% RSLogix 500 project INVENTORY_MANAGEMENT.RSS, saved by version 8.30.00.16 %
PROJECT "UNTITLED"    % processor: Bul.1763 MicroLogix 1100 Series B %

PROGRAM FILES
  LAD 2 "MAIN"  6 rungs
  LAD 3 "EXTRACT"  7 rungs
  LAD 4 "COMPUTE"  4 rungs
  LAD 5 "CLEAR"  2 rungs

DATA FILES
  O0 OUTPUT  4 elements
  I1 INPUT  6 elements
  S2 STATUS  66 elements
  B3 BINARY  1 elements
  T4 TIMER  1 elements
  C5 COUNTER  1 elements
  R6 CONTROL  1 elements
  N7 INTEGER  6 elements
  F8 FLOAT  1 elements
  N9 SCN_BUFFER  4 elements
  ST10 STRING  5 elements

LADDER 2 "MAIN"
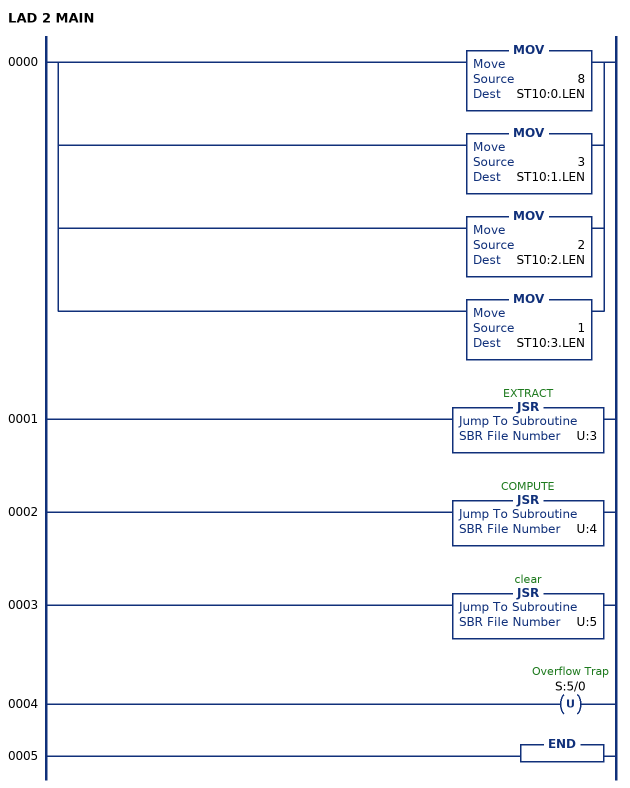
% Rung: 0 %
SOR BST MOV 8 ST10:0.LEN NXB MOV 3 ST10:1.LEN NXB MOV 2 ST10:2.LEN NXB MOV 1 ST10:3.LEN BND EOR
% Rung: 1 %
SOR JSR U:3 EOR
%   U:3  "EXTRACT" %
% Rung: 2 %
SOR JSR U:4 EOR
%   U:4  "COMPUTE" %
% Rung: 3 %
SOR JSR U:5 EOR
%   U:5  "clear" %
% Rung: 4 %
SOR OTU S:5/0 EOR
%   S:5/0  "Overflow Trap" %
% Rung: 5 %
SOR END EOR

LADDER 3 "EXTRACT"
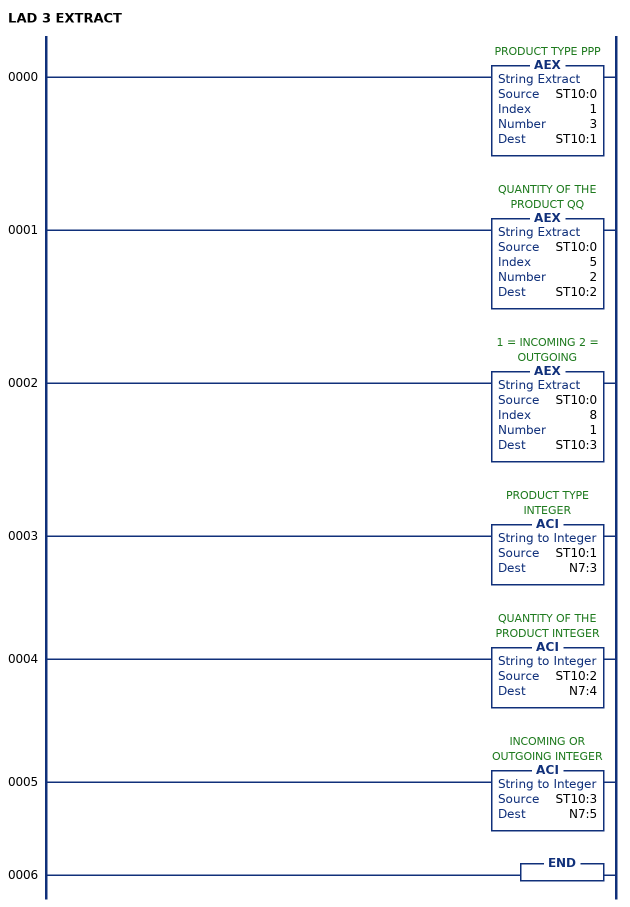
% Rung: 0 %
SOR AEX ST10:0 1 3 ST10:1 EOR
%   ST10:0  "SCANNED CODE AS STRING" %
%   ST10:1  "PRODUCT TYPE PPP" %
% Rung: 1 %
SOR AEX ST10:0 5 2 ST10:2 EOR
%   ST10:0  "SCANNED CODE AS STRING" %
%   ST10:2  "QUANTITY OF THE PRODUCT QQ" %
% Rung: 2 %
SOR AEX ST10:0 8 1 ST10:3 EOR
%   ST10:0  "SCANNED CODE AS STRING" %
%   ST10:3  "1 = INCOMING 2 = OUTGOING" %
% Rung: 3 %
SOR ACI ST10:1 N7:3 EOR
%   ST10:1  "PRODUCT TYPE PPP" %
%   N7:3  "PRODUCT TYPE INTEGER" %
% Rung: 4 %
SOR ACI ST10:2 N7:4 EOR
%   ST10:2  "QUANTITY OF THE PRODUCT QQ" %
%   N7:4  "QUANTITY OF THE PRODUCT INTEGER" %
% Rung: 5 %
SOR ACI ST10:3 N7:5 EOR
%   ST10:3  "1 = INCOMING 2 = OUTGOING" %
%   N7:5  "INCOMING OR OUTGOING INTEGER" %
% Rung: 6 %
SOR END EOR

LADDER 4 "COMPUTE"
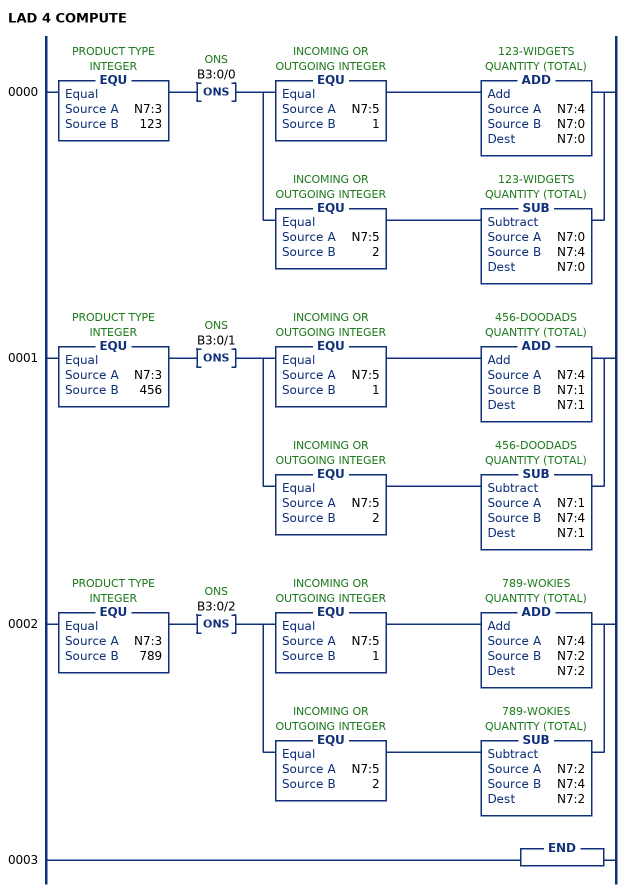
% Rung: 0 %
SOR EQU N7:3 123 ONS B3:0/0 BST EQU N7:5 1 ADD N7:4 N7:0 N7:0 NXB EQU N7:5 2 SUB N7:0 N7:4 N7:0 BND EOR
%   N7:3  "PRODUCT TYPE INTEGER" %
%   B3:0/0  "ONS" %
%   N7:5  "INCOMING OR OUTGOING INTEGER" %
%   N7:4  "QUANTITY OF THE PRODUCT INTEGER" %
%   N7:0  "123-WIDGETS QUANTITY (TOTAL)" %
% Rung: 1 %
SOR EQU N7:3 456 ONS B3:0/1 BST EQU N7:5 1 ADD N7:4 N7:1 N7:1 NXB EQU N7:5 2 SUB N7:1 N7:4 N7:1 BND EOR
%   N7:3  "PRODUCT TYPE INTEGER" %
%   B3:0/1  "ONS" %
%   N7:5  "INCOMING OR OUTGOING INTEGER" %
%   N7:4  "QUANTITY OF THE PRODUCT INTEGER" %
%   N7:1  "456-DOODADS QUANTITY (TOTAL)" %
% Rung: 2 %
SOR EQU N7:3 789 ONS B3:0/2 BST EQU N7:5 1 ADD N7:4 N7:2 N7:2 NXB EQU N7:5 2 SUB N7:2 N7:4 N7:2 BND EOR
%   N7:3  "PRODUCT TYPE INTEGER" %
%   B3:0/2  "ONS" %
%   N7:5  "INCOMING OR OUTGOING INTEGER" %
%   N7:4  "QUANTITY OF THE PRODUCT INTEGER" %
%   N7:2  "789-WOKIES QUANTITY (TOTAL)" %
% Rung: 3 %
SOR END EOR

LADDER 5 "CLEAR"
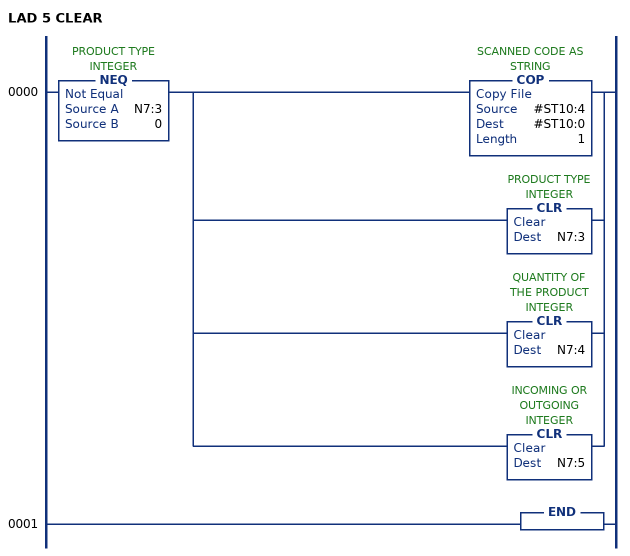
% Rung: 0 %
SOR NEQ N7:3 0 BST COP #ST10:4 #ST10:0 1 NXB CLR N7:3 NXB CLR N7:4 NXB CLR N7:5 BND EOR
%   N7:3  "PRODUCT TYPE INTEGER" %
%   ST10:4  "empty string" %
%   ST10:0  "SCANNED CODE AS STRING" %
%   N7:4  "QUANTITY OF THE PRODUCT INTEGER" %
%   N7:5  "INCOMING OR OUTGOING INTEGER" %
% Rung: 1 %
SOR END EOR

OTHER DOCUMENTED ADDRESSES
  ST10:0.0  "Length of the Scanned Code"
  ST10:0.1  "DATA FROM THE SCANNER"

DATA TABLE (non-zero values as saved)
DATA ST10
% ST10:0 % "0"
% ST10:1 % "0"
% ST10:2 % "0"
% ST10:3 % "0"
